PROGRAM P_StablePlatform
VAR
	fbpA 		: FB_AnalogInputScaling;
	fbpB 		: FB_AnalogInputScaling;
	fbpS 	 	: FB_AnalogInputScaling;
	fSVFeedback : FB_AnalogInputScaling;
	fbPistonPos	: FB_AnalogInputScaling_1;
	fbPistonVel	: FB_AnalogInputScaling_1;
	fbJoystick  : FB_JoystickInputScaling;
	fbSVOutput 	: FB_ValveOutput;
	bManualMode : BOOL;
END_VAR

// Inputs
fbpA(
	nRawInput := G_StablePlatformIO.npA,
	stAnalogInputScaling := G_StablePlatformParameters.stPressureSensorScaling400bar,
	fOutput => G_StablePlatformScaledIO.bpA
);

fbpB(
	nRawInput := G_StablePlatformIO.npB,
	stAnalogInputScaling := G_StablePlatformParameters.stPressureSensorScaling400bar,
	fOutput => G_StablePlatformScaledIO.bpB
);

fbpS(
	nRawInput := G_StablePlatformIO.npS,
	stAnalogInputScaling := G_StablePlatformParameters.stPressureSensorScaling400bar,
	fOutput => G_StablePlatformScaledIO.bpS
);

fSVFeedback(
	nRawInput := G_StablePlatformIO.nSVFeedback,
	stAnalogInputScaling := G_StablePlatformParameters.stSVFeedbackScaling,
	fOutput => G_StablePlatformScaledIO.fSVFeedback
);


fbJoystick(
	bEnable := bManualMode,
	nRawInput := G_Inputs.stJoyLX.nValue,
	stJoystickInputScaling := G_StablePlatformParameters.stJoystickInputScalingX,
	fNormalizedOutput => G_StablePlatformScaledIO.fJoystickNormalizedX
);

// Outputs
fbSVOutput(
	bEnable := G_Inputs.bJoystickLeftEnable AND bManualMode,
	bDeadBandCompOn := FALSE,
	stValveDeadBand := G_StablePlatformParameters.stSVValveDeadBand,
	fNormalizedInput := -G_StablePlatformScaledIO.fJoystickNormalizedX,
	nOutput => G_StablePlatformIO.nSVControlSignal
);

G_StablePlatformIO.bSVEnable := bManualMode;

fbPistonPos(
	nRawInput := G_StablePlatformIO.nPistonPosition,
	stAnalogInputScaling := G_StablePlatformParameters.stPistonPos,
	fOutput => G_StablePlatformScaledIO.fPistonPosition
);

fbPistonVel(
	nRawInput := G_StablePlatformIO.nPistonVelocity,
	stAnalogInputScaling := G_StablePlatformParameters.stPistonVel,
	fOutput => G_StablePlatformScaledIO.fPistonPosition
);

G_StablePlatformParameters.fPlatformAngle := fPlatformAngleTheta1(G_StablePlatformScaledIO.fPistonPosition);

END_PROGRAM

(* stored: Version 1.1.0.1, ProductVersion 3.1.4024.12
   POU P_StablePlatform: Id {c20de7b0-d2cd-4536-8a51-2764cdc32403}, SpecialFunc None *)
